% RSLogix 500 project motor_forward_reverse_basic.RSS, saved by version 8.30.00.16 %
PROJECT "FORREV"    % processor: Bul.1763 MicroLogix 1100 Series B %

PROGRAM FILES
  LAD 2   5 rungs

DATA FILES
  O0 OUTPUT  4 elements
  I1 INPUT  6 elements
  S2 STATUS  66 elements
  B3 BINARY  1 elements
  T4 TIMER  1 elements
  C5 COUNTER  1 elements
  R6 CONTROL  1 elements
  N7 INTEGER  1 elements
  F8 FLOAT  1 elements

LADDER 2
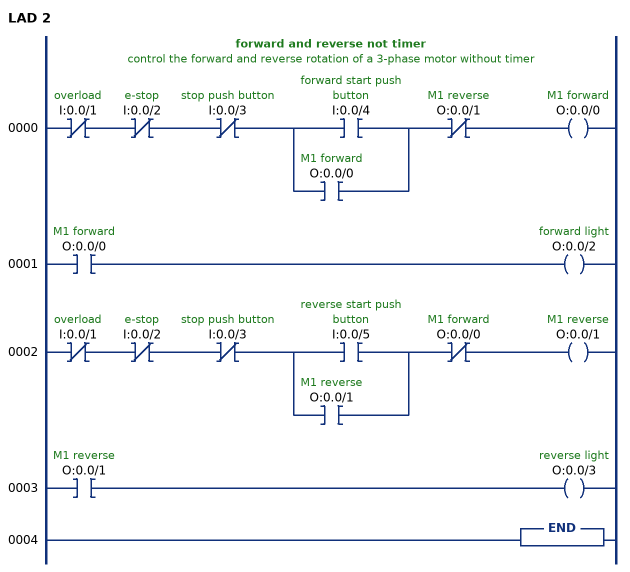
% Rung: 0 %
% TITLE: forward and reverse not timer %
% control the forward and reverse rotation of a 3-phase motor without timer %
SOR XIO I:0.0/1 XIO I:0.0/2 XIO I:0.0/3 BST XIC I:0.0/4 NXB XIC O:0.0/0 BND XIO O:0.0/1 OTE O:0.0/0 EOR
%   I:0.0/1  "overload" %
%   I:0.0/2  "e-stop" %
%   I:0.0/3  "stop push button" %
%   I:0.0/4  "forward start push button" %
%   O:0.0/0  "M1 forward" %
%   O:0.0/1  "M1 reverse" %
% Rung: 1 %
SOR XIC O:0.0/0 OTE O:0.0/2 EOR
%   O:0.0/0  "M1 forward" %
%   O:0.0/2  "forward light" %
% Rung: 2 %
SOR XIO I:0.0/1 XIO I:0.0/2 XIO I:0.0/3 BST XIC I:0.0/5 NXB XIC O:0.0/1 BND XIO O:0.0/0 OTE O:0.0/1 EOR
%   I:0.0/1  "overload" %
%   I:0.0/2  "e-stop" %
%   I:0.0/3  "stop push button" %
%   I:0.0/5  "reverse start push button" %
%   O:0.0/1  "M1 reverse" %
%   O:0.0/0  "M1 forward" %
% Rung: 3 %
SOR XIC O:0.0/1 OTE O:0.0/3 EOR
%   O:0.0/1  "M1 reverse" %
%   O:0.0/3  "reverse light" %
% Rung: 4 %
SOR END EOR
